// TIA Portal V18 export
ORGANIZATION_BLOCK "Main"   // OB1, LAD, ProgramCycle
TITLE = "Main Program Sweep (Cycle)"
{ S7_Optimized_Access := 'TRUE' }
VERSION : 0.1
// stored: AutoNumber true, IsIECCheckEnabled false, SetENOAutomatically false
   VAR_INPUT
      Initial_Call : Bool;   // Initial call of this OB
      Remanence : Bool;   // =True, if remanent data are available
   END_VAR
BEGIN

REGION Network 1: Вже вiдпрацьовано?
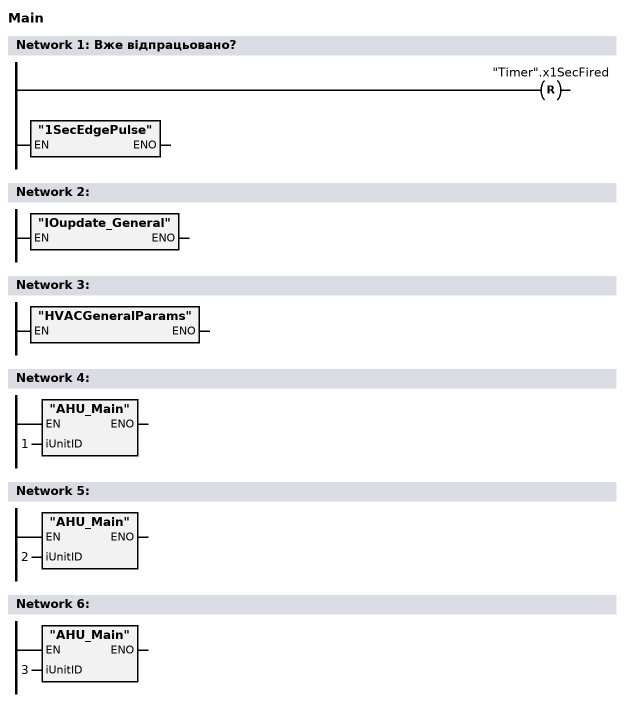
   RUNG wire#powerrail
      R_Coil( "Timer".x1SecFired )
   END_RUNG
   RUNG wire#powerrail
      "1SecEdgePulse"()
   END_RUNG
   // the same network as SCL:
   "Timer".x1SecFired := FALSE;
   "1SecEdgePulse"();
END_REGION

REGION Network 2
   RUNG wire#powerrail
      "IOupdate_General"()
   END_RUNG
   // the same network as SCL:
   "IOupdate_General"();
END_REGION

REGION Network 3
   RUNG wire#powerrail
      "HVACGeneralParams"()
   END_RUNG
   // the same network as SCL:
   "HVACGeneralParams"();
END_REGION

REGION Network 4
   RUNG wire#powerrail
      "AHU_Main"(iUnitID := 1)
   END_RUNG
   // the same network as SCL:
   "AHU_Main"(iUnitID := 1);
END_REGION

REGION Network 5
   RUNG wire#powerrail
      "AHU_Main"(iUnitID := 2)
   END_RUNG
   // the same network as SCL:
   "AHU_Main"(iUnitID := 2);
END_REGION

REGION Network 6
   RUNG wire#powerrail
      "AHU_Main"(iUnitID := 3)
   END_RUNG
   // the same network as SCL:
   "AHU_Main"(iUnitID := 3);
END_REGION

REGION Network 10 (SCL)
   //CASE "Calculated_VariablesF".ModeFromPanel OF
   //    0:  // OFF
   //        "AO_1".FanModulation := 0.0 ;
   //    2:  // Speed1
   //        "AO_1".FanModulation := "Seted_VariablesF".SAFSpeed1;
   //    3:  // Speed2     
   //        "AO_1".FanModulation := "Seted_VariablesF".SAFSpeed2;
   //    ELSE  // Auto
   //        "AO_1".FanModulation := "Seted_VariablesF".SAFSpeedAuto;
   //END_CASE;
END_REGION
END_ORGANIZATION_BLOCK
